Staubli VAL3: Frame.pjx

--- Frame.pjx ---
Parameters version=s7.8.3 stackSize=5000 millimeterUnit=true
Program file=Edit.pgx
Program file=EnterPageKey.pgx
Program file=getFrame.pgx
Program file=Main.pgx
Program file=MainKey.pgx
Program file=OnF1.pgx
Program file=OnF2.pgx
Program file=OnF7.pgx
Program file=OnF8.pgx
Program file=Refresh.pgx
Program file=RefreshList.pgx
Program file=SetFrame.pgx
Program file=start.pgx
Program file=stop.pgx
Data file=Frame.dtx
Library alias=user path=Disk://userPage/USERPAGE.pjx

--- Frame.dtx ---
bool bExit
bool bListRefresh
bool bUserRefresh
public frame fFrame{}
  [Frame1] = {x=480, y=190, z=-101.4, rx=2, rz=-90, fatherId=world[0]}
  [Frame10] = {fatherId=world[0]}
  [Frame11] = {fatherId=world[0]}
  [Frame12] = {fatherId=world[0]}
  [Frame13] = {fatherId=world[0]}
  [Frame14] = {fatherId=world[0]}
  [Frame15] = {fatherId=world[0]}
  [Frame16] = {fatherId=world[0]}
  [Frame17] = {fatherId=world[0]}
  [Frame18] = {fatherId=world[0]}
  [Frame19] = {fatherId=world[0]}
  [Frame2] = {fatherId=world[0]}
  [Frame20] = {fatherId=world[0]}
  [Frame3] = {fatherId=world[0]}
  [Frame4] = {fatherId=world[0]}
  [Frame5] = {fatherId=world[0]}
  [Frame6] = {fatherId=world[0]}
  [Frame7] = {fatherId=world[0]}
  [Frame8] = {fatherId=world[0]}
  [Frame9] = {fatherId=world[0]}
mdesc mNomSpeed
num nSelected
num nType
string sFrameName
string sItem
string sList
string sListItemValue
string sParameter

--- Main.pgx ---
public program Main(num x_nType)
  local num l_nKey
begin
  //
  bUserRefresh=bListRefresh=true
  bExit=false
  nType=x_nType
  //
  do
    call Refresh()
    call RefreshList()
    call user:setList("坐标系",sList,bUserRefresh,bListRefresh,nSelected,sItem,l_nKey)
    bUserRefresh=false
    bListRefresh=false
    call MainKey(l_nKey)
    delay(0)
  until bExit

end

--- start.pgx ---
public program start()
begin
  call Main(0)
end

--- Edit.pgx ---
program Edit()
  local bool l_bRes
  local num l_i
  local string l_sValue
  local num l_nSelect
  local string l_sItem
  local num l_nKey
  local num l_nRes
begin

  cls()
  resize(sParameter,1,6)
  sParameter[0]="X"
  sParameter[1]="Y"
  sParameter[2]="Z"
  sParameter[3]="Rx"
  sParameter[4]="Ry"
  sParameter[5]="Rz"
  //
  resize(sListItemValue,1,size(sParameter))
  sListItemValue[0]=toString(".3",fFrame[sItem].trsf.x)
  sListItemValue[1]=toString(".3",fFrame[sItem].trsf.y)
  sListItemValue[2]=toString(".3",fFrame[sItem].trsf.z)
  sListItemValue[3]=toString(".3",fFrame[sItem].trsf.rx)
  sListItemValue[4]=toString(".3",fFrame[sItem].trsf.ry)
  sListItemValue[5]=toString(".3",fFrame[sItem].trsf.rz)
  //
  for l_i=0 to size(sParameter)-1
    call user:strlength(sParameter[l_i],user:nBottomX/2)
    l_sValue=sListItemValue[l_i]
    call user:strlength(l_sValue,user:nBottomX/2+1)
    sParameter[l_i]=sParameter[l_i]+":"+l_sValue
  endFor

  bUserRefresh=true
  bListRefresh=true
  //
  do
    if bUserRefresh
      cls()
      call user:clear(0,13)
      call user:typeMenu(8,"确定")
    endIf
    call user:setList(sItem,sParameter,bUserRefresh,bListRefresh,l_nSelect,l_sItem,l_nKey)
    bUserRefresh=false
    bListRefresh=false
    call EnterPageKey(l_nKey,l_nSelect,sParameter[l_nSelect])
    delay(0)
  until l_nKey==255 or l_nKey==278
  bUserRefresh=true
  bListRefresh=true
end

--- EnterPageKey.pgx ---
program EnterPageKey(num& x_nKey, num& x_nSelect, string& x_sItem)
  local string l_sStr
  local num l_nKey
  local string l_sEmpty
  local string l_sValue
  local num l_nItem
  local num l_nView
  local string l_sItem
  local point lp
  local string l_sYN[2]
  local bool l_bRes
begin
  //
  switch x_nSelect
    case 0
      if x_nKey==270
        call user:editNum(x_sItem,sListItemValue[x_nSelect],fFrame[sItem].trsf.x,x_nSelect)
      endIf
    break
    case 1
      if x_nKey==270
        call user:editNum(x_sItem,sListItemValue[x_nSelect],fFrame[sItem].trsf.y,x_nSelect)
      endIf
    break
    case 2
      if x_nKey==270
         call user:editNum(x_sItem,sListItemValue[x_nSelect],fFrame[sItem].trsf.z,x_nSelect)
      endIf
    break
    case 3
      if x_nKey==270
        call user:editNum(x_sItem,sListItemValue[x_nSelect],fFrame[sItem].trsf.rx,x_nSelect)
      endIf
    break
    case 4
      if x_nKey==27
         call user:editNum(x_sItem,sListItemValue[x_nSelect],fFrame[sItem].trsf.ry,x_nSelect)
      endIf
    break
    case 5
      if x_nKey==270
        call user:editNum(x_sItem,sListItemValue[x_nSelect],fFrame[sItem].trsf.rz,x_nSelect)
      endIf
    break
  endSwitch
  if x_nKey==270
    bUserRefresh=true
    bListRefresh=true
  endIf
end

--- getFrame.pgx ---
public program getFrame(string& x_sFrm, frame& x_fFrame)
begin
  x_sFrm=sFrameName
  x_fFrame.trsf=fFrame[sFrameName].trsf
end

--- OnF1.pgx ---
program OnF1()
begin
  if nType==1
    call SetFrame(sItem)
    popUpMsg("选择坐标系："+sItem)
  endIf
end

--- OnF2.pgx ---
program OnF2()
begin
  call Edit()
end

--- Refresh.pgx ---
program Refresh()
begin
  //
  if bUserRefresh
    cls()
    userPage()
    if nType==1
      gotoxy(1,1)
      put("F1->确定")
      gotoxy(1,13)
      put("F1")
    endIf

    gotoxy(1,2)
    put("F2->编辑")
    gotoxy(6,13)
    put("F2")
    //    gotoxy(1,3)
    //    put("F3->删除")
    //    gotoxy(11,13)
    //    put("F3")
    //    gotoxy(1,4)
    //    put("F4->编辑路径")
    //    gotoxy(16,13)
    //    put("编辑")
    //
    //    gotoxy(1,6)
    //    put("F6->")
    //    gotoxy(26,13)
    //    put("")
    gotoxy(1,7)
    put("F7->保存")
    gotoxy(31,13)
    put("F7")
    gotoxy(1,8)
    put("F8->返回")
    gotoxy(36,13)
    put("F8")
  endIf
end

--- RefreshList.pgx ---
program RefreshList()
  local num l_ni
begin
  //
  if bListRefresh
    resize(sList,1,20)
    for l_ni=0 to 19
      sList[l_ni]="Frame"+toString("",l_ni+1)
    endFor
  endIf

end

--- SetFrame.pgx ---
public program SetFrame(string x_sFrame)
begin
  //
  sFrameName=x_sFrame
end
